VAR_GLOBAL PERSISTENT
	arrPalette					: ARRAY [0..200] OF ST_Dut_Data;
END_VAR

(* stored: Version 1.1.0.1, ProductVersion 3.1.4024.12
   GVL GVL_Palette: Id {c71107be-0c8b-4ca9-99f8-358fcf99acf0} *)
